PROGRAM MAIN
VAR
	//Train function
    Train : treinrit;
END_VAR

CASE gvl.Step OF

    0: (* Start at home *)
        gvl.sStatus := 'leaving home, get in the car, driving to station';
        gvl.bStartDrive := TRUE;
        gvl.tDriveHomeToStation(IN := gvl.bStartDrive);

        IF gvl.tDriveHomeToStation.Q THEN
            gvl.bStartDrive := FALSE;
            gvl.tDriveHomeToStation(IN := FALSE);
            gvl.Step := 5;
        END_IF;


    5: (* Walking from car to train*)
        gvl.sStatus := 'parked the car. Walking to the station.';
        gvl.bStartWalk1 := TRUE;
        gvl.tWalkHomeToStation(IN := gvl.bStartWalk1);

        IF gvl.tWalkHomeToStation.Q THEN
            gvl.bStartWalk1 := FALSE;
            gvl.tWalkHomeToStation(IN := FALSE);
            gvl.Step := 10;
        END_IF;


    10: (* Start train*)
        gvl.sStatus := 'Aarrived at the station. Train leaves.';
        gvl.bStartTrain := TRUE;
        Train(Start := gvl.bStartTrain, TravelTime := T#12S);

        IF Train.Arrived THEN
            gvl.bStartTrain := FALSE;
            gvl.Step := 20;
        END_IF;


    20: (* Walking from train to school *)
        gvl.sStatus := 'Train arrived. Walking to school.';
        gvl.bStartWalk2 := TRUE;
        gvl.tWalkStationToSchool(IN := gvl.bStartWalk2);

        IF gvl.tWalkStationToSchool.Q THEN
            gvl.tWalkStationToSchool(IN := FALSE);
            gvl.bStartWalk2 := FALSE;
            gvl.Step := 30;
        END_IF;


    30: (* Arrived at school *)
        gvl.sStatus := 'arrived at school';


ELSE
    gvl.sStatus := 'ERROR, I am lost.';
END_CASE;

END_PROGRAM

(* stored: Version 1.1.0.1, ProductVersion 3.1.4024.15
   POU MAIN: Id {7724f42e-4414-46f2-83ac-ecbdc8010cf1}, SpecialFunc None *)
